PROGRAM PRG_OverridePressure
VAR
	fb_SetPressure : FB_SetChamberPressure; 
END_VAR

fb_SetPressure(chamber := stVl_Proto, rNewPressure := New_Pressure, Override:= Global_OverridePressure);

END_PROGRAM

(* stored: Version 1.1.0.1, ProductVersion 3.1.4022.12
   POU PRG_OverridePressure: Id {21e5fc14-89ca-42fb-9669-1519ab1832f3}, SpecialFunc None *)
